(* PLC project Tank, Unknown Tank 1 *)
(* stored: creationDateTime 2026-08-17T12:00:00, modificationDateTime 2026-08-19T18:25:52 *)

FUNCTION_BLOCK TempCtrl
  VAR_INPUT
    Temp : INT;  (* Measured milk temperature *)
    Setpoint : INT;  (* pasteurization target *)
    Inhibit : BOOL;  (* if TRUE, force heat to 0 (dry-fire interlock) *)
  END_VAR
  VAR_OUTPUT
    Power : INT;  (* heater command 0-100% *)
  END_VAR
  VAR
    out : REAL;  (* computed heater power 0-100 *)
    err : REAL;  (* setpoint minus measured temperature *)
    integ : REAL;  (* integral accumulator (with anti-windup) *)
    KP : REAL;  (* proportional gain *)
    KI : REAL;  (* integral gain per second *)
  END_VAR

            (* PI heater control with anti-windup.
   err > 0 means the milk is too cold -> call for heat. *)
  KP := 8.0;
  KI := 1.5;
  err := INT_TO_REAL(Setpoint) - INT_TO_REAL(Temp);

  (* provisional output = proportional + accumulated integral *)
  out := KP * err + integ;

  (* ANTI-WINDUP: only grow the integral while we are NOT saturated.
     Climbing from cold, out is pinned at 100%, so we freeze the
     integral instead of letting it wind up past the setpoint. *)
  IF (out > 0.0) AND (out < 100.0) THEN
      integ := integ + KI * err * 0.02;   (* 0.02 s = the 20 ms scan *)
  END_IF;

  out := LIMIT(0.0, KP * err + integ, 100.0);

  (* dry-fire / phase interlock: force heat off and drop the integral *)
  IF Inhibit THEN
      out   := 0.0;
      integ := 0.0;
  END_IF;

  Power := REAL_TO_INT(out);

          
END_FUNCTION_BLOCK

PROGRAM program0
  VAR
    Temperature AT %QW0 : INT;  (* Measured milk temperature in the vat (deg C). Written by the plant; read by the PLC. *)
    Level AT %QW1 : INT;  (* Measured milk level in the vat (percent full). Written by the plant; read by the PLC. *)
    TempSetpoint AT %QW2 : INT;  (* Operator pasteurization target temperature (deg C, nominally 63). *)
    HoldSecs AT %QW5 : INT;  (* time *)
    LevelSetpoint AT %QW3 : INT;  (* Operator target fill level (percent). *)
    Heater AT %QX0.0 : BOOL;  (* STATUS lamp: TRUE when HeaterPower > 0 (the jacket is calling for heat). Read by the HMI. *)
    Pump AT %QX0.1 : BOOL;  (* Command to the fill pump. On during the Fill phase; forced off while Emptying. *)
    AlmPastTemp AT %QX0.2 : BOOL;  (* CRITICAL ALARM: while cooking, milk is below the pasteurization setpoint. *)
    AlmHighTemp AT %QX0.3 : BOOL;  (* ALARM: milk temperature above the safe band (scorch). *)
    AlmLowLevel AT %QX0.4 : BOOL;  (* ALARM: vat level below 20 percent. Dry-fire risk; inhibits the heater. *)
    AlmHighLevel AT %QX0.5 : BOOL;  (* ALARM: vat level above 90 percent. Overflow risk. *)
    BatchSafe AT %QX0.6 : BOOL;  (* TRUE when milk was held at/above setpoint for the full hold time. Pasteurized. *)
    Divert AT %QX0.7 : BOOL;  (* Fail-safe reject. TRUE whenever the batch is not proven safe (NOT BatchSafe). *)
    Discharge AT %QX1.0 : BOOL;  (* Discharge valve. Open only during the Empty phase (Emptying). *)
    HeaterPower AT %QW4 : INT;  (* PI heater command 0-100 percent. Written by the PLC; read by the plant. *)
  END_VAR
  VAR
    AtTemp : BOOL;  (* Internal: TRUE when Temperature >= TempSetpoint. *)
    TankFull : BOOL;  (* Internal: TRUE when Level >= LevelSetpoint (vat filled). *)
    TankEmpty : BOOL;  (* Internal: TRUE when Level <= 3 (vat drained). *)
    Cooking : BOOL;  (* STATE latch: heat+hold phase. Set at TankFull, reset by Emptying. *)
    Emptying : BOOL;  (* STATE latch: discharge phase. Set at BatchSafe, reset by TankEmpty. *)
    HeatInhibit : BOOL;  (* Internal: AlmLowLevel OR NOT Cooking. Feeds the TempCtrl Inhibit (heat only while cooking). *)
    BelowSP : BOOL;  (* Internal: TRUE when Temperature < TempSetpoint. Used by AlmPastTemp. *)
    LevelLow : BOOL;  (* Internal: pump hysteresis LOW flag (Level < LevelLowInt). *)
    LevelHigh : BOOL;  (* Internal: pump hysteresis HIGH flag (Level > LevelHighInt). *)
    LevelLowInt : INT;  (* Internal: LevelSetpoint - 5. *)
    LevelHighInt : INT;  (* Internal: LevelSetpoint + 5. *)
    TempHiThr : INT;  (* Internal: TempSetpoint + 5 (overheat alarm threshold). *)
    HoldTimer : TON;  (* Internal hold timer. IN = AtTemp AND Cooking, PT = T#30s. Q sets BatchSafe. *)
    TempCtrl0 : TempCtrl;  (* Instance of the PI temperature-control function block. *)
  END_VAR

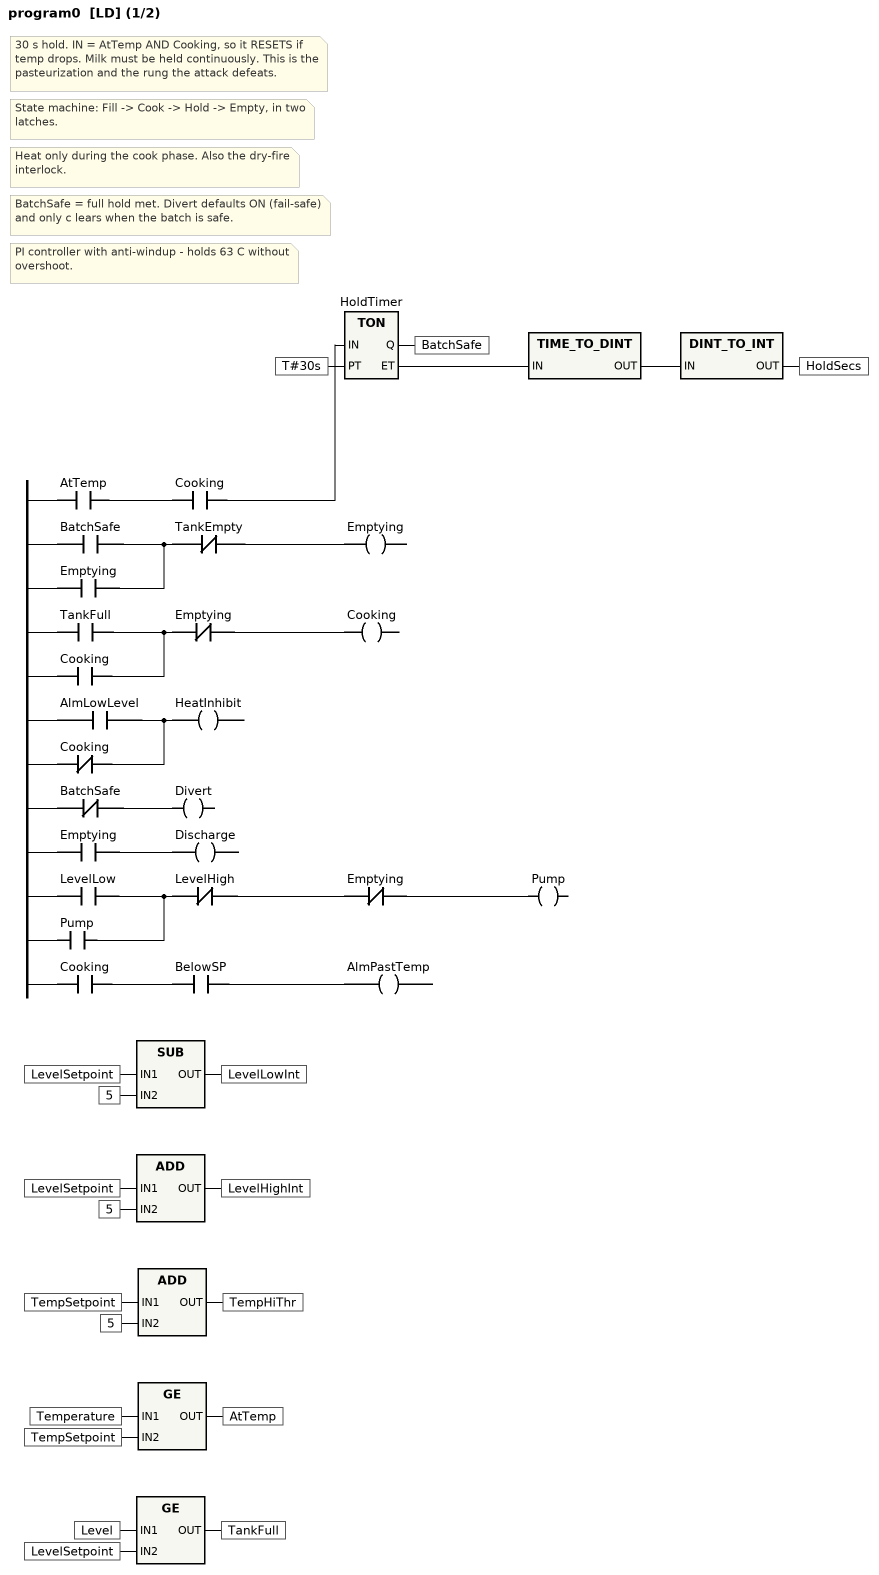
(* LD diagram, written out as Structured Text *)
LevelLowInt := LevelSetpoint - 5;
LevelHighInt := LevelSetpoint + 5;
TempHiThr := TempSetpoint + 5;
AtTemp := Temperature >= TempSetpoint;
TankFull := Level >= LevelSetpoint;
TankEmpty := Level <= 3;
AlmLowLevel := Level < 20;
AlmHighLevel := Level > 90;
AlmHighTemp := Temperature > TempHiThr;
BelowSP := Temperature < TempSetpoint;
LevelLow := Level < LevelLowInt;
LevelHigh := Level > LevelHighInt;
Heater := HeaterPower > 0;
(* PI controller with anti-windup - holds 63 C without overshoot. *)
(* 30 s hold. IN = AtTemp AND Cooking, so it RESETS if temp drops. Milk must be held continuously. This is the pasteurization and the rung the attack defeats. *)
TempCtrl0(Temp := Temperature, Setpoint := TempSetpoint, Inhibit := HeatInhibit);
HeaterPower := TempCtrl0.Power;
HoldTimer(IN := AtTemp AND Cooking, PT := T#30s);
BatchSafe := HoldTimer.Q;
Emptying := (BatchSafe OR Emptying) AND NOT TankEmpty;
(* State machine: Fill -> Cook -> Hold -> Empty, in two latches. *)
Cooking := (TankFull OR Cooking) AND NOT Emptying;
(* Heat only during the cook phase. Also the dry-fire interlock. *)
HeatInhibit := AlmLowLevel OR NOT Cooking;
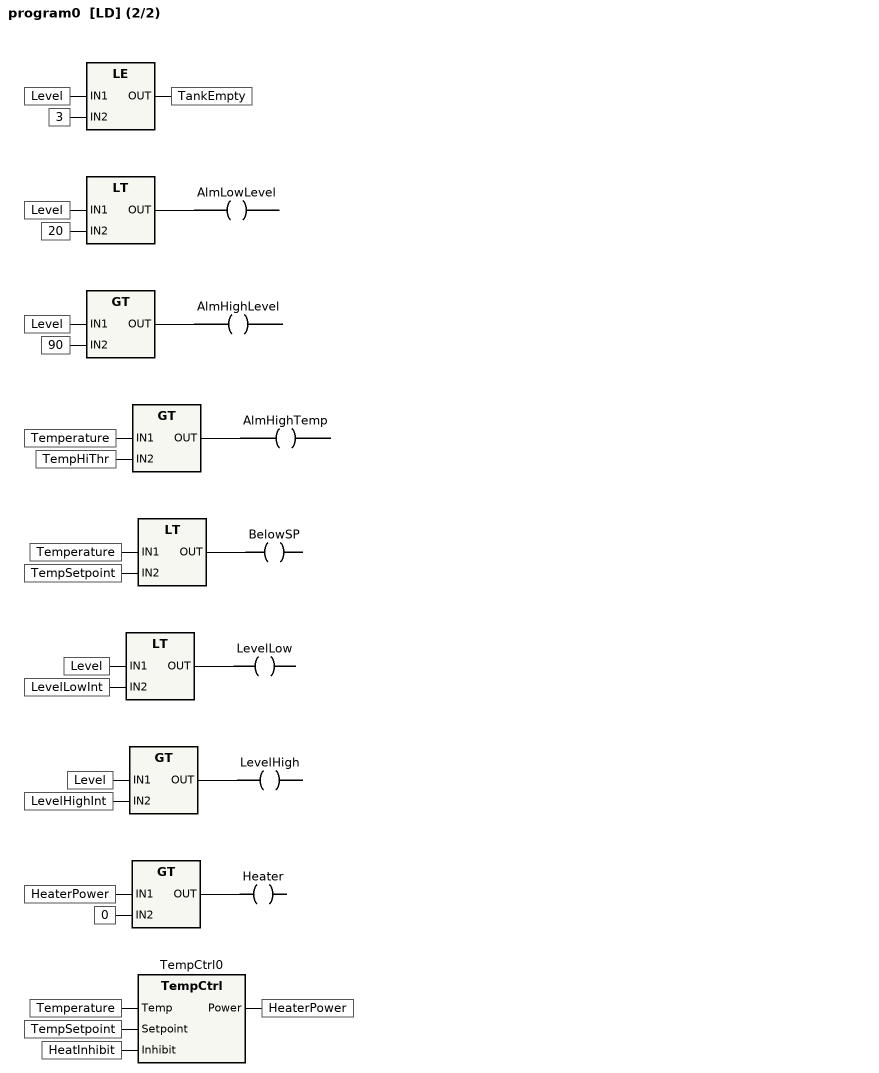
Divert := NOT BatchSafe;
(* BatchSafe = full hold met. Divert defaults ON (fail-safe) and only c lears when the batch is safe. *)
Discharge := Emptying;
Pump := (LevelLow OR Pump) AND NOT LevelHigh AND NOT Emptying;
AlmPastTemp := Cooking AND BelowSP;
HoldSecs := DINT_TO_INT(TIME_TO_DINT(HoldTimer.ET));
END_PROGRAM

CONFIGURATION Config0
  RESOURCE Res0 ON PLC
    TASK task0(INTERVAL := T#20ms, PRIORITY := 0);
    PROGRAM instance0 WITH task0 : program0;
  END_RESOURCE
END_CONFIGURATION
